{attribute 'linkalways'} 
{attribute 'no_explicit_call' := 'This FB is a CLASS and must be accessed using methods or properties'}
{attribute 'enable_dynamic_creation'}
FUNCTION_BLOCK _ETcVnPrototypeClusterer EXTENDS EnumDatatypeBase
VAR
	localData : ETcVnPrototypeClusterer;
	activeData : REFERENCE TO ETcVnPrototypeClusterer;
	enumBaseDatatype : _UDINT(localData);
END_VAR

METHOD PRIVATE AddLocalEnumeration
VAR_INPUT
	Enumeration : T_MAXSTRING;
	Value : ETcVnPrototypeClusterer;
END_VAR
AddEnumeration(Enumeration, Value);
END_METHOD

PROPERTY PUBLIC Address : PVOID
GET
Address := ADR(activeData);
END_GET
END_PROPERTY

METHOD PUBLIC ClearReference
VAR_INPUT
END_VAR
activeData REF= localData;
SetBaseDatatypeReference();
END_METHOD

METHOD PUBLIC Clone : I_Datatype
VAR
    pClone : POINTER TO _ETcVnPrototypeClusterer;
END_VAR
pClone := __NEW(_ETcVnPrototypeClusterer(InitialValue := Value));
Clone := pClone^;
END_METHOD

METHOD FB_init : BOOL
VAR_INPUT
	bInitRetains : BOOL; // if TRUE, the retain variables are initialized (warm start / cold start)
	bInCopyCode : BOOL;  // if TRUE, the instance afterwards gets moved into the copy code (online change)
	InitialValue : ETcVnPrototypeClusterer;
END_VAR
localData := InitialValue;
AddBaseDatatype(enumBaseDatatype);
ClearReference();

AddLocalEnumeration('TCVN_PC_NOVELTY_DETECTOR', ETcVnPrototypeClusterer.TCVN_PC_NOVELTY_DETECTOR);
AddLocalEnumeration('TCVN_PC_CLUSTERER', ETcVnPrototypeClusterer.TCVN_PC_CLUSTERER);
END_METHOD

PROPERTY PUBLIC Identifier : T_MAXSTRING
GET
Identifier := 'ETcVnPrototypeClusterer';
END_GET
END_PROPERTY

METHOD IsEnumeratorValueEqual : BOOL
VAR_INPUT
	Enumerator : I_KeyValueForwardEnumerator;
END_VAR
VAR
	storedValue : ETcVnPrototypeClusterer;
END_VAR
IF NOT Enumerator.TryGet(storedValue) THEN
	RETURN;
END_IF

IsEnumeratorValueEqual := storedValue = activeData;
END_METHOD

METHOD PUBLIC MakeReferenceTo
VAR_INPUT
	ReferenceTarget : REFERENCE TO ETcVnPrototypeClusterer;
END_VAR
activeData REF= ReferenceTarget;
SetBaseDatatypeReference();
END_METHOD

METHOD PROTECTED SetBaseDatatypeReference
VAR_INPUT
END_VAR
enumBaseDatatype.MakeReferenceTo(activeData);
END_METHOD

PROPERTY PUBLIC Size : UDINT
GET
Size := SIZEOF(activeData);
END_GET
END_PROPERTY

METHOD TryMakeReferenceTo : BOOL
VAR_INPUT
	Target : I_Datatype;
END_VAR
VAR
	targetAsEnum : I_EnumDatatype;
	pTargetData : POINTER TO ETcVnPrototypeClusterer;
END_VAR
IF NOT Target.TryResolveAsEnumDatatype(targetAsEnum) THEN
	RETURN;
END_IF

IF targetAsEnum.Identifier <> Identifier THEN
	RETURN;
END_IF

pTargetData := Target.Address;
activeData REF= pTargetData^;
SetBaseDatatypeReference();
TryMakeReferenceTo := TRUE;
END_METHOD

PROPERTY PUBLIC Value : ETcVnPrototypeClusterer
GET
Value := activeData;
END_GET
SET
activeData := Value;
END_SET
END_PROPERTY

END_FUNCTION_BLOCK

(* stored: Version 1.1.0.1
   POU _ETcVnPrototypeClusterer: Id {a88e5ac5-cc26-4e5b-87c3-641e5102617f}, SpecialFunc None
   Folder Constructor: Id {6c8c98f9-d05f-45cd-81ab-0c26fc7a9174}
   Folder Private: Id {8054ad65-cff8-4542-8bd7-5267a4d2750a}
   Folder Protected: Id {4be3f8af-15d6-4906-80a6-9a059030f080}
   Method AddLocalEnumeration: Id {85a62aa4-784f-43e7-9dc2-5ac1395c2c34}
   Property Address: Id {6774d1d6-8383-4b8e-be11-234bc74c702b}
   Get Get: Id {29972928-345e-404d-81f3-a833381c01fb}
   Method ClearReference: Id {a8c6e5ca-aa16-4435-a3a7-acebe59ceeb5}
   Method Clone: Id {7a594cf4-397e-4953-b75c-5f18b1df64f3}
   Method FB_init: Id {06c3199d-2d6f-4ed5-9672-9916c88de741}
   Property Identifier: Id {9d6b3a10-1931-4fd5-a838-41a9ca380cc8}
   Get Get: Id {d7bed805-27d3-45a3-939d-796ddff9ae3c}
   Method IsEnumeratorValueEqual: Id {36637acc-f8c7-445b-bcac-6d90c6a13428}
   Method MakeReferenceTo: Id {913df407-8cbe-4854-8196-d645b5870575}
   Method SetBaseDatatypeReference: Id {0c821452-3189-44ce-8766-9f3f635ec809}
   Property Size: Id {ec5b35fa-a1bb-4e18-a7e0-8d0ec04b5e6c}
   Get Get: Id {8110ca94-c3a9-44d5-b3dd-23b9e0247efb}
   Method TryMakeReferenceTo: Id {89b0fe7f-7100-40c9-8186-dabd9ff09ab0}
   Property Value: Id {810d5829-d32a-4d98-b454-697cbfd59cf7}
   Get Get: Id {54ab3b4c-39b9-470f-818a-60f527044fbc}
   Set Set: Id {8c48dd33-5e0b-4092-931f-964162ea32ef} *)
